// TIA Portal V20 export
FUNCTION "PMC_Config_Map00" : Void   // FC121, LAD
// stored: Namespace CITI_Logic, SetENOAutomatically false
BEGIN

REGION Network 1: Remote Config_En
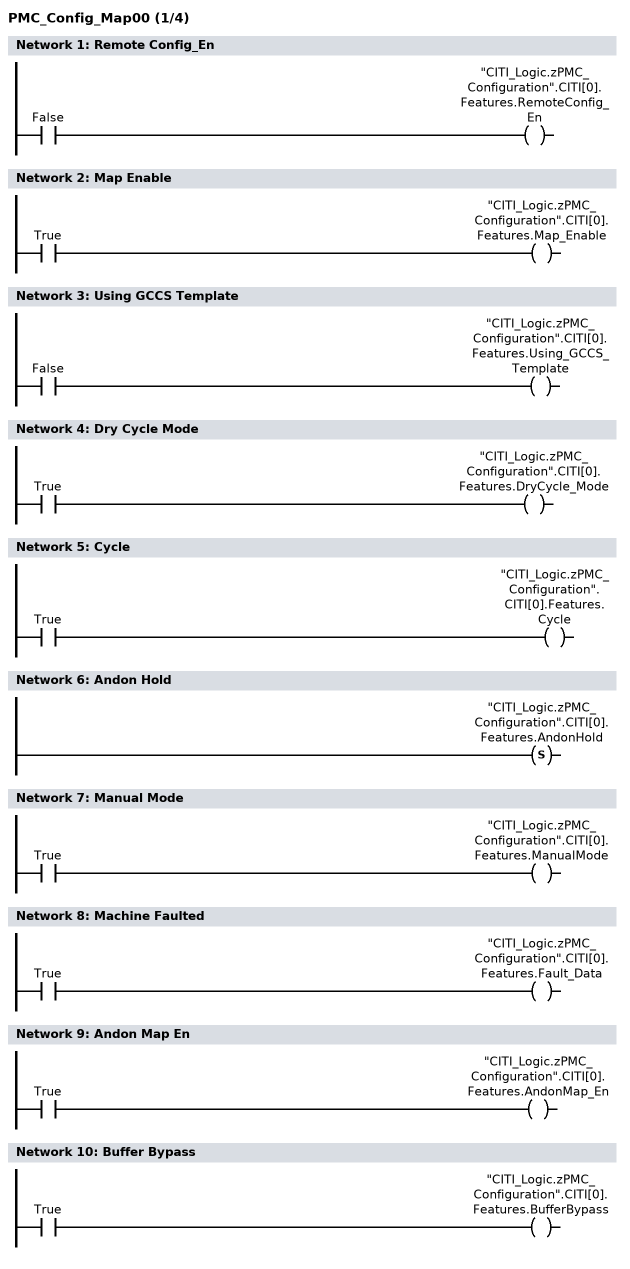
   RUNG wire#powerrail
      Contact( False )
      Coil( "CITI_Logic.zPMC_Configuration".CITI[0].Features.RemoteConfig_En )
   END_RUNG
   // the same network as SCL:
   "CITI_Logic.zPMC_Configuration".CITI[0].Features.RemoteConfig_En := False;
END_REGION

REGION Network 2: Map Enable
   RUNG wire#powerrail
      Contact( True )
      Coil( "CITI_Logic.zPMC_Configuration".CITI[0].Features.Map_Enable )
   END_RUNG
   // the same network as SCL:
   "CITI_Logic.zPMC_Configuration".CITI[0].Features.Map_Enable := True;
END_REGION

REGION Network 3: Using GCCS Template
   RUNG wire#powerrail
      Contact( False )
      Coil( "CITI_Logic.zPMC_Configuration".CITI[0].Features.Using_GCCS_Template )
   END_RUNG
   // the same network as SCL:
   "CITI_Logic.zPMC_Configuration".CITI[0].Features.Using_GCCS_Template := False;
END_REGION

REGION Network 4: Dry Cycle Mode
   RUNG wire#powerrail
      Contact( True )
      Coil( "CITI_Logic.zPMC_Configuration".CITI[0].Features.DryCycle_Mode )
   END_RUNG
   // the same network as SCL:
   "CITI_Logic.zPMC_Configuration".CITI[0].Features.DryCycle_Mode := True;
END_REGION

REGION Network 5: Cycle
   RUNG wire#powerrail
      Contact( True )
      Coil( "CITI_Logic.zPMC_Configuration".CITI[0].Features.Cycle )
   END_RUNG
   // the same network as SCL:
   "CITI_Logic.zPMC_Configuration".CITI[0].Features.Cycle := True;
END_REGION

REGION Network 6: Andon Hold
   RUNG wire#powerrail
      S_Coil( "CITI_Logic.zPMC_Configuration".CITI[0].Features.AndonHold )
   END_RUNG
   // the same network as SCL:
   "CITI_Logic.zPMC_Configuration".CITI[0].Features.AndonHold := TRUE;
END_REGION

REGION Network 7: Manual Mode
   RUNG wire#powerrail
      Contact( True )
      Coil( "CITI_Logic.zPMC_Configuration".CITI[0].Features.ManualMode )
   END_RUNG
   // the same network as SCL:
   "CITI_Logic.zPMC_Configuration".CITI[0].Features.ManualMode := True;
END_REGION

REGION Network 8: Machine Faulted
   RUNG wire#powerrail
      Contact( True )
      Coil( "CITI_Logic.zPMC_Configuration".CITI[0].Features.Fault_Data )
   END_RUNG
   // the same network as SCL:
   "CITI_Logic.zPMC_Configuration".CITI[0].Features.Fault_Data := True;
END_REGION

REGION Network 9: Andon Map En
   RUNG wire#powerrail
      Contact( True )
      Coil( "CITI_Logic.zPMC_Configuration".CITI[0].Features.AndonMap_En )
   END_RUNG
   // the same network as SCL:
   "CITI_Logic.zPMC_Configuration".CITI[0].Features.AndonMap_En := True;
END_REGION

REGION Network 10: Buffer Bypass
   RUNG wire#powerrail
      Contact( True )
      Coil( "CITI_Logic.zPMC_Configuration".CITI[0].Features.BufferBypass )
   END_RUNG
   // the same network as SCL:
   "CITI_Logic.zPMC_Configuration".CITI[0].Features.BufferBypass := True;
END_REGION

REGION Network 11: Bypass
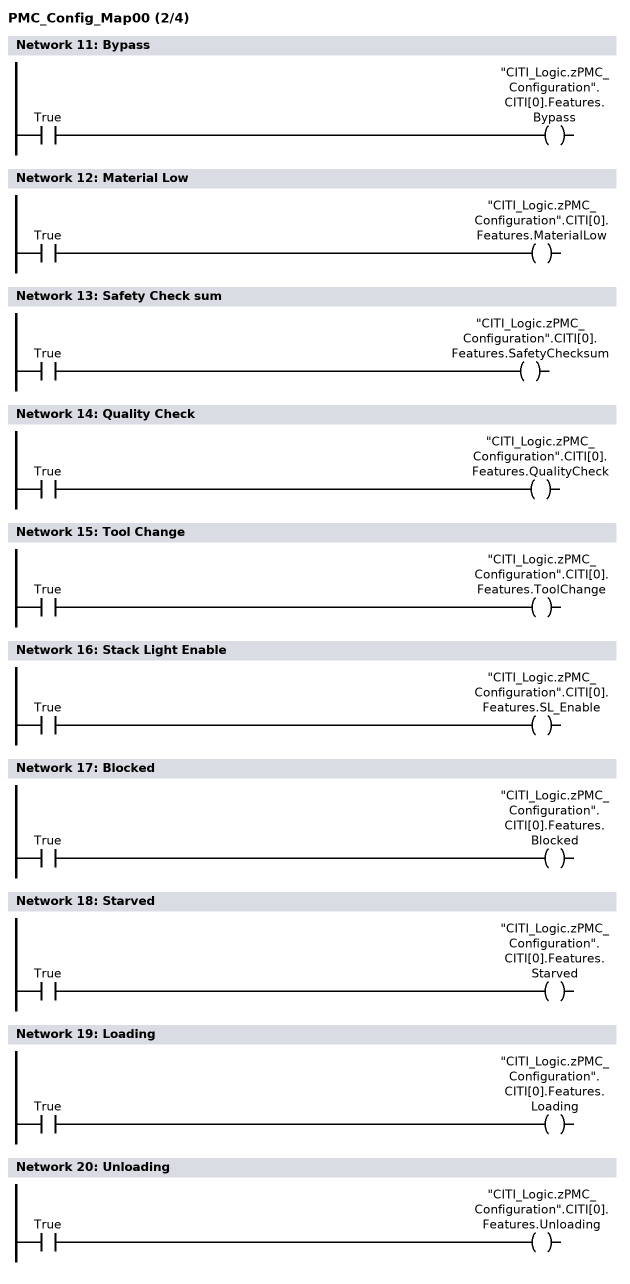
   RUNG wire#powerrail
      Contact( True )
      Coil( "CITI_Logic.zPMC_Configuration".CITI[0].Features.Bypass )
   END_RUNG
   // the same network as SCL:
   "CITI_Logic.zPMC_Configuration".CITI[0].Features.Bypass := True;
END_REGION

REGION Network 12: Material Low
   RUNG wire#powerrail
      Contact( True )
      Coil( "CITI_Logic.zPMC_Configuration".CITI[0].Features.MaterialLow )
   END_RUNG
   // the same network as SCL:
   "CITI_Logic.zPMC_Configuration".CITI[0].Features.MaterialLow := True;
END_REGION

REGION Network 13: Safety Check sum
   RUNG wire#powerrail
      Contact( True )
      Coil( "CITI_Logic.zPMC_Configuration".CITI[0].Features.SafetyChecksum )
   END_RUNG
   // the same network as SCL:
   "CITI_Logic.zPMC_Configuration".CITI[0].Features.SafetyChecksum := True;
END_REGION

REGION Network 14: Quality Check
   RUNG wire#powerrail
      Contact( True )
      Coil( "CITI_Logic.zPMC_Configuration".CITI[0].Features.QualityCheck )
   END_RUNG
   // the same network as SCL:
   "CITI_Logic.zPMC_Configuration".CITI[0].Features.QualityCheck := True;
END_REGION

REGION Network 15: Tool Change
   RUNG wire#powerrail
      Contact( True )
      Coil( "CITI_Logic.zPMC_Configuration".CITI[0].Features.ToolChange )
   END_RUNG
   // the same network as SCL:
   "CITI_Logic.zPMC_Configuration".CITI[0].Features.ToolChange := True;
END_REGION

REGION Network 16: Stack Light Enable
   RUNG wire#powerrail
      Contact( True )
      Coil( "CITI_Logic.zPMC_Configuration".CITI[0].Features.SL_Enable )
   END_RUNG
   // the same network as SCL:
   "CITI_Logic.zPMC_Configuration".CITI[0].Features.SL_Enable := True;
END_REGION

REGION Network 17: Blocked
   RUNG wire#powerrail
      Contact( True )
      Coil( "CITI_Logic.zPMC_Configuration".CITI[0].Features.Blocked )
   END_RUNG
   // the same network as SCL:
   "CITI_Logic.zPMC_Configuration".CITI[0].Features.Blocked := True;
END_REGION

REGION Network 18: Starved
   RUNG wire#powerrail
      Contact( True )
      Coil( "CITI_Logic.zPMC_Configuration".CITI[0].Features.Starved )
   END_RUNG
   // the same network as SCL:
   "CITI_Logic.zPMC_Configuration".CITI[0].Features.Starved := True;
END_REGION

REGION Network 19: Loading
   RUNG wire#powerrail
      Contact( True )
      Coil( "CITI_Logic.zPMC_Configuration".CITI[0].Features.Loading )
   END_RUNG
   // the same network as SCL:
   "CITI_Logic.zPMC_Configuration".CITI[0].Features.Loading := True;
END_REGION

REGION Network 20: Unloading
   RUNG wire#powerrail
      Contact( True )
      Coil( "CITI_Logic.zPMC_Configuration".CITI[0].Features.Unloading )
   END_RUNG
   // the same network as SCL:
   "CITI_Logic.zPMC_Configuration".CITI[0].Features.Unloading := True;
END_REGION

REGION Network 21: Idle
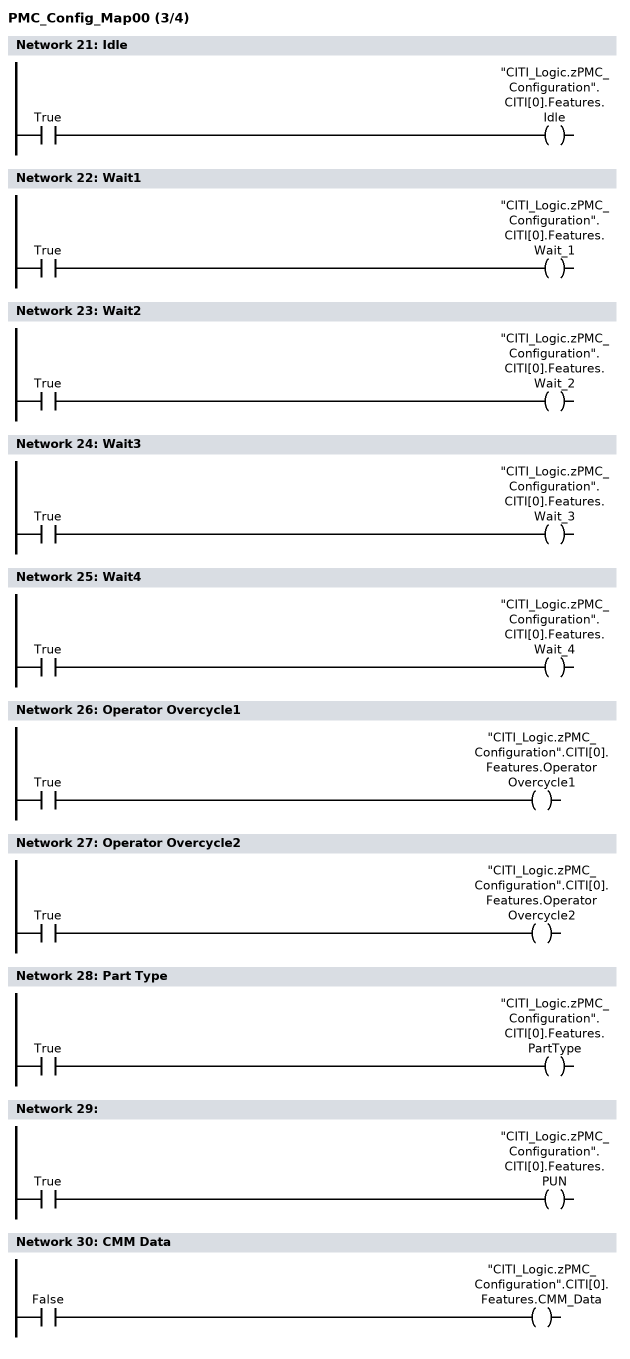
   RUNG wire#powerrail
      Contact( True )
      Coil( "CITI_Logic.zPMC_Configuration".CITI[0].Features.Idle )
   END_RUNG
   // the same network as SCL:
   "CITI_Logic.zPMC_Configuration".CITI[0].Features.Idle := True;
END_REGION

REGION Network 22: Wait1
   RUNG wire#powerrail
      Contact( True )
      Coil( "CITI_Logic.zPMC_Configuration".CITI[0].Features.Wait_1 )
   END_RUNG
   // the same network as SCL:
   "CITI_Logic.zPMC_Configuration".CITI[0].Features.Wait_1 := True;
END_REGION

REGION Network 23: Wait2
   RUNG wire#powerrail
      Contact( True )
      Coil( "CITI_Logic.zPMC_Configuration".CITI[0].Features.Wait_2 )
   END_RUNG
   // the same network as SCL:
   "CITI_Logic.zPMC_Configuration".CITI[0].Features.Wait_2 := True;
END_REGION

REGION Network 24: Wait3
   RUNG wire#powerrail
      Contact( True )
      Coil( "CITI_Logic.zPMC_Configuration".CITI[0].Features.Wait_3 )
   END_RUNG
   // the same network as SCL:
   "CITI_Logic.zPMC_Configuration".CITI[0].Features.Wait_3 := True;
END_REGION

REGION Network 25: Wait4
   RUNG wire#powerrail
      Contact( True )
      Coil( "CITI_Logic.zPMC_Configuration".CITI[0].Features.Wait_4 )
   END_RUNG
   // the same network as SCL:
   "CITI_Logic.zPMC_Configuration".CITI[0].Features.Wait_4 := True;
END_REGION

REGION Network 26: Operator Overcycle1
   RUNG wire#powerrail
      Contact( True )
      Coil( "CITI_Logic.zPMC_Configuration".CITI[0].Features.OperatorOvercycle1 )
   END_RUNG
   // the same network as SCL:
   "CITI_Logic.zPMC_Configuration".CITI[0].Features.OperatorOvercycle1 := True;
END_REGION

REGION Network 27: Operator Overcycle2
   RUNG wire#powerrail
      Contact( True )
      Coil( "CITI_Logic.zPMC_Configuration".CITI[0].Features.OperatorOvercycle2 )
   END_RUNG
   // the same network as SCL:
   "CITI_Logic.zPMC_Configuration".CITI[0].Features.OperatorOvercycle2 := True;
END_REGION

REGION Network 28: Part Type
   RUNG wire#powerrail
      Contact( True )
      Coil( "CITI_Logic.zPMC_Configuration".CITI[0].Features.PartType )
   END_RUNG
   // the same network as SCL:
   "CITI_Logic.zPMC_Configuration".CITI[0].Features.PartType := True;
END_REGION

REGION Network 29
   RUNG wire#powerrail
      Contact( True )
      Coil( "CITI_Logic.zPMC_Configuration".CITI[0].Features.PUN )
   END_RUNG
   // the same network as SCL:
   "CITI_Logic.zPMC_Configuration".CITI[0].Features.PUN := True;
END_REGION

REGION Network 30: CMM Data
   RUNG wire#powerrail
      Contact( False )
      Coil( "CITI_Logic.zPMC_Configuration".CITI[0].Features.CMM_Data )
   END_RUNG
   // the same network as SCL:
   "CITI_Logic.zPMC_Configuration".CITI[0].Features.CMM_Data := False;
END_REGION

REGION Network 31: Filter Data
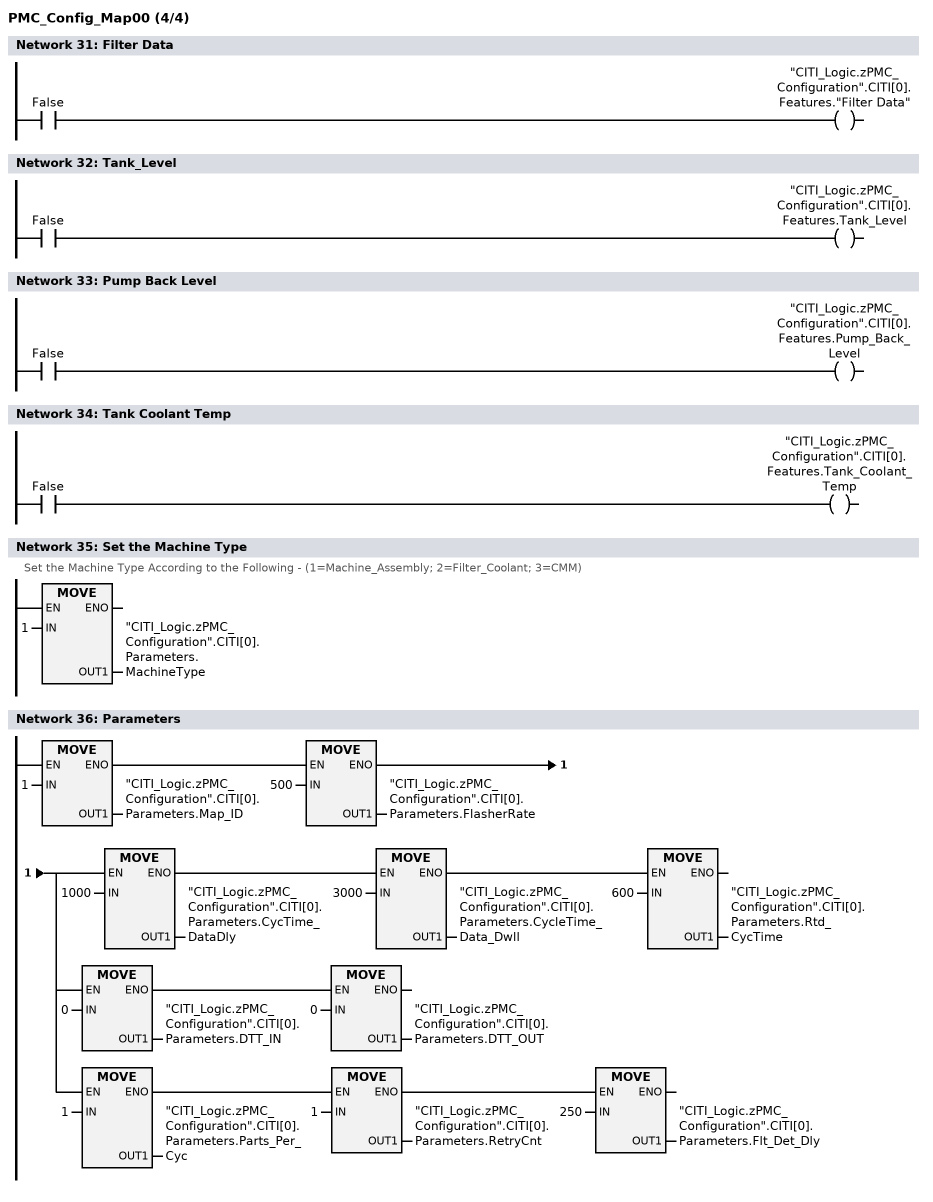
   RUNG wire#powerrail
      Contact( False )
      Coil( "CITI_Logic.zPMC_Configuration".CITI[0].Features."Filter Data" )
   END_RUNG
   // the same network as SCL:
   "CITI_Logic.zPMC_Configuration".CITI[0].Features."Filter Data" := False;
END_REGION

REGION Network 32: Tank_Level
   RUNG wire#powerrail
      Contact( False )
      Coil( "CITI_Logic.zPMC_Configuration".CITI[0].Features.Tank_Level )
   END_RUNG
   // the same network as SCL:
   "CITI_Logic.zPMC_Configuration".CITI[0].Features.Tank_Level := False;
END_REGION

REGION Network 33: Pump Back Level
   RUNG wire#powerrail
      Contact( False )
      Coil( "CITI_Logic.zPMC_Configuration".CITI[0].Features.Pump_Back_Level )
   END_RUNG
   // the same network as SCL:
   "CITI_Logic.zPMC_Configuration".CITI[0].Features.Pump_Back_Level := False;
END_REGION

REGION Network 34: Tank Coolant Temp
   RUNG wire#powerrail
      Contact( False )
      Coil( "CITI_Logic.zPMC_Configuration".CITI[0].Features.Tank_Coolant_Temp )
   END_RUNG
   // the same network as SCL:
   "CITI_Logic.zPMC_Configuration".CITI[0].Features.Tank_Coolant_Temp := False;
END_REGION

REGION Network 35: Set the Machine Type
   // Set the Machine Type According to the Following - (1=Machine_Assembly; 2=Filter_Coolant; 3=CMM)
   RUNG wire#powerrail
      Move(in := 1, out1 => "CITI_Logic.zPMC_Configuration".CITI[0].Parameters.MachineType)
   END_RUNG
   // the same network as SCL:
   "CITI_Logic.zPMC_Configuration".CITI[0].Parameters.MachineType := 1;
END_REGION

REGION Network 36: Parameters
   RUNG wire#powerrail
      Move(in := 1, out1 => "CITI_Logic.zPMC_Configuration".CITI[0].Parameters.Map_ID)
      Move(in := 500, out1 => "CITI_Logic.zPMC_Configuration".CITI[0].Parameters.FlasherRate)
      wire#w1
      Move(in := 1000, out1 => "CITI_Logic.zPMC_Configuration".CITI[0].Parameters.CycTime_DataDly)
      Move(in := 3000, out1 => "CITI_Logic.zPMC_Configuration".CITI[0].Parameters.CycleTime_Data_Dwll)
      Move(in := 600, out1 => "CITI_Logic.zPMC_Configuration".CITI[0].Parameters.Rtd_CycTime)
   END_RUNG
   RUNG wire#w1
      Move(in := 0, out1 => "CITI_Logic.zPMC_Configuration".CITI[0].Parameters.DTT_IN)
      Move(in := 0, out1 => "CITI_Logic.zPMC_Configuration".CITI[0].Parameters.DTT_OUT)
   END_RUNG
   RUNG wire#w1
      Move(in := 1, out1 => "CITI_Logic.zPMC_Configuration".CITI[0].Parameters.Parts_Per_Cyc)
      Move(in := 1, out1 => "CITI_Logic.zPMC_Configuration".CITI[0].Parameters.RetryCnt)
      Move(in := 250, out1 => "CITI_Logic.zPMC_Configuration".CITI[0].Parameters.Flt_Det_Dly)
   END_RUNG
   // the same network as SCL:
   "CITI_Logic.zPMC_Configuration".CITI[0].Parameters.Map_ID := 1;
   "CITI_Logic.zPMC_Configuration".CITI[0].Parameters.FlasherRate := 500;
   "CITI_Logic.zPMC_Configuration".CITI[0].Parameters.CycTime_DataDly := 1000;
   "CITI_Logic.zPMC_Configuration".CITI[0].Parameters.CycleTime_Data_Dwll := 3000;
   "CITI_Logic.zPMC_Configuration".CITI[0].Parameters.Rtd_CycTime := 600;
   "CITI_Logic.zPMC_Configuration".CITI[0].Parameters.DTT_IN := 0;
   "CITI_Logic.zPMC_Configuration".CITI[0].Parameters.DTT_OUT := 0;
   "CITI_Logic.zPMC_Configuration".CITI[0].Parameters.Parts_Per_Cyc := 1;
   "CITI_Logic.zPMC_Configuration".CITI[0].Parameters.RetryCnt := 1;
   "CITI_Logic.zPMC_Configuration".CITI[0].Parameters.Flt_Det_Dly := 250;
END_REGION
END_FUNCTION
